TYPE ST_DeviceStateTable :
STRUCT
	iDeviceID:DINT;
	iStateID:DINT;
	rTargetPosition: REAL;
	rTolerance: REAL;
	rTransmission: REAL;
	iBeamClass : DINT;
	rPhotonEnergy: REAL;
END_STRUCT
END_TYPE

(* stored: Version 1.1.0.1, ProductVersion 3.1.4022.12
   DUT ST_DeviceStateTable: Id {03fca704-e94f-069c-15d5-ec1df795b0de} *)
